(***********************************************************************************************************************************************
*********** OUTPUT FHPP DATA *******************************************************************************************************************
***********************************************************************************************************************************************)

pFHPP_DATA_OUT				:= ADR(FML_REF.FHPP.OUT);

IF FML_REF.Modbus THEN				// modbus word swapping
	//first 8 Byte
	FHPP_Target[0]			:= pFHPP_DATA_OUT^[1];
	FHPP_Target[1]			:= pFHPP_DATA_OUT^[0];
	FHPP_Target[2]			:= pFHPP_DATA_OUT^[3];
	FHPP_Target[3]			:= pFHPP_DATA_OUT^[2];
	IF FML_REF.HighByteFirst THEN	// high byte first (actual value2)
		FHPP_Target[4]		:= pFHPP_DATA_OUT^[6];
		FHPP_Target[5]		:= pFHPP_DATA_OUT^[7];
		FHPP_Target[6]		:= pFHPP_DATA_OUT^[4];
		FHPP_Target[7]		:= pFHPP_DATA_OUT^[5];
	ELSE							// low byte first (actual value2)
		FHPP_Target[4]		:= pFHPP_DATA_OUT^[5];
		FHPP_Target[5]		:= pFHPP_DATA_OUT^[4];
		FHPP_Target[6]		:= pFHPP_DATA_OUT^[7];
		FHPP_Target[7]		:= pFHPP_DATA_OUT^[6];
	END_IF	
	
	//second 8 Byte
	FHPP_Target[8]			:= pFHPP_DATA_OUT^[9];
	FHPP_Target[9]			:= pFHPP_DATA_OUT^[8];
	FHPP_Target[10]			:= pFHPP_DATA_OUT^[11];
	FHPP_Target[11]			:= pFHPP_DATA_OUT^[10];
	IF FML_REF.HighByteFirst THEN	// high byte first (actual value2)
		FHPP_Target[12]		:= pFHPP_DATA_OUT^[14];
		FHPP_Target[13]		:= pFHPP_DATA_OUT^[15];
		FHPP_Target[14]		:= pFHPP_DATA_OUT^[12];
		FHPP_Target[15]		:= pFHPP_DATA_OUT^[13];
	ELSE							// low byte first (actual value2)
		FHPP_Target[12]		:= pFHPP_DATA_OUT^[13];
		FHPP_Target[13]		:= pFHPP_DATA_OUT^[12];
		FHPP_Target[14]		:= pFHPP_DATA_OUT^[15];
		FHPP_Target[15]		:= pFHPP_DATA_OUT^[14];
	END_IF	
	
ELSE								//normal fieldbus: copy only
	// first 8 byte
	FHPP_Target[0]			:= pFHPP_DATA_OUT^[0];
	FHPP_Target[1]			:= pFHPP_DATA_OUT^[1];
	FHPP_Target[2]			:= pFHPP_DATA_OUT^[2];
	FHPP_Target[3]			:= pFHPP_DATA_OUT^[3];
	IF FML_REF.HighByteFirst THEN	// high byte first (actual value2)
		FHPP_Target[4]		:= pFHPP_DATA_OUT^[7];
		FHPP_Target[5]		:= pFHPP_DATA_OUT^[6];
		FHPP_Target[6]		:= pFHPP_DATA_OUT^[5];
		FHPP_Target[7]		:= pFHPP_DATA_OUT^[4];
	ELSE							// low byte first (actual value2)
		FHPP_Target[4]		:= pFHPP_DATA_OUT^[4];
		FHPP_Target[5]		:= pFHPP_DATA_OUT^[5];
		FHPP_Target[6]		:= pFHPP_DATA_OUT^[6];
		FHPP_Target[7]		:= pFHPP_DATA_OUT^[7];
	END_IF	
	
	// second 8 byte
	FHPP_Target[8]			:= pFHPP_DATA_OUT^[8];
	FHPP_Target[9]			:= pFHPP_DATA_OUT^[9];
	FHPP_Target[10]			:= pFHPP_DATA_OUT^[10];
	FHPP_Target[11]			:= pFHPP_DATA_OUT^[11];
	IF FML_REF.HighByteFirst THEN	// high byte first (actual value2)
		FHPP_Target[12]		:= pFHPP_DATA_OUT^[15];
		FHPP_Target[13]		:= pFHPP_DATA_OUT^[14];
		FHPP_Target[14]		:= pFHPP_DATA_OUT^[13];
		FHPP_Target[15]		:= pFHPP_DATA_OUT^[12];
	ELSE							// low byte first (actual value2)
		FHPP_Target[12]		:= pFHPP_DATA_OUT^[12];
		FHPP_Target[13]		:= pFHPP_DATA_OUT^[13];
		FHPP_Target[14]		:= pFHPP_DATA_OUT^[14];
		FHPP_Target[15]		:= pFHPP_DATA_OUT^[15];
	END_IF	
END_IF

(* ===== end of function block ============================= *)

END_FUNCTION_BLOCK

// Blocks/Parameterize/FPC_DATA_OBJECT
(* ============================================================================
   FESTO AG  Co., Esslingen - Copyright (c) 2015. All rights reserved.                       
 ------------------------------------------------------------------------------
 Functionblock:  FPC_DATA_OBJECT  
 Description:    function block to pass internal data objects to the controller
 Version:        V3.5.4.4        
 Composer:       bejk
 Last Update:    13.11.2017                                                                           
 ------------------------------------------------------------------------------ *)
{library private}
(* ----------------------------------------------------------------------------
Date        Name                Activity                                                                              
02.02.2010  Benjamin Kilgus     created
02.07.2013  Rudolf Schenke      Busy state and some other value clear
22.06.2015	Christian Hammer	adaptation to use this FB for all drives
04.09.2015  Christian Hammer	error handling (deleted RETVAL, created Status)
29.02.2016	Christian Hammer	set outputs to zero if not execute
13.11.2017	Christian Hammer	added blockade of FB for SFC-DC and MTR-DCI controller
=============================================================================== *)
{library public}

(* use this function block only with the function blocks FML_Read and FML_Write *)

FUNCTION_BLOCK FPC_DATA_OBJECT

VAR_IN_OUT
	FML_REF				: DT_FML_REF;		// structure of the parameter to control and parametrize the motorcontroller
END_VAR

VAR_INPUT
	Execute				: BOOL;  			// perfrom data exchange
	Write				: BOOL;  			// read or write the parameter (1=write / 0=read)
	Object				: INT; 				// number of internal data object
	Subindex			: INT; 				// subindex of the parameter to exchange
	Value				: DINT; 			// set value of internal data objects
END_VAR
VAR_OUTPUT
	Done				: BOOL; 			// transmission done
	Error				: BOOL; 			// transmission fault
	Status				: DT_FML_STATUS;	// structure with the status information of the function block and FPC
	ActObject			: INT;				// actual number of internal data objects
	ActSubindex			: DINT; 			// actual subindex of the parameter
	ActValue			: DINT; 			// actual value of internal data objects	
END_VAR

{library private}
VAR
	bInit           	: BOOL	:=FALSE;	// status of inizialisation of the FB
	lMemberID   		: INT;				// local member ID of the FB
	Step				: INT	:= 0;		// step number of the state machine

	TONInst				: TON;				// timer instance to monitor a timeout of the function block
	TimeStart			: BOOL;				// variable to start the timer instance
	TimeoutTime			: TIME := T#3S;		// timeout time 			
END_VAR
{library public}

(* ====== initial block routine ===================================== *)
(* ----- get MemberID for this function block ------------------------*)

IF NOT bInit THEN
	FML_REF.MemberIDmax		:= FML_REF.MemberIDmax +1;
	lMemberID				:= FML_REF.MemberIDmax;
	bInit					:= TRUE;
	Status.Err:=FALSE; Status.Cat:=FML_function_block; Status.ID:=FML_init_active;
END_IF

	
(* ====== supervision of timeout ==================================== *)
(* ----- timer to monitor a timeout of the function block ------------*)
TONInst(IN := TimeStart, PT := TimeoutTime);
IF TONInst.Q THEN
	Status.Err:=TRUE; Status.Cat:=FML_function_block; Status.ID:=FML_fb_timeout;
	Done					:= TRUE;
	Step					:= 100;
END_IF		

// this function block is not usable with SFC-DC and MTR-DCI
IF Execute 
	AND	((FML_REF.DeviceType = SFC_DC)
	OR (FML_REF.DeviceType = MTR_DCI)) THEN
		Done				:= TRUE;
		Status.Err:=TRUE; Status.Cat:=FML_function_block; Status.ID:=FML_wrong_device;
		Step				:= 100;
END_IF

(* ===== logic part ================================================= *)

IF NOT Execute AND (Step <> 0) THEN
 	FML_REF.MemberID		:= 0;
	FML_REF.ReqID			:= FML_FPC_REQ_none;
	FML_REF.FPCC_Modus		:= 0;
	FML_REF.PNU				:= 0;
	FML_REF.Subindex		:= 0;
	FML_REF.Value			:= 0;
	ActObject				:= 0;
	ActSubindex				:= 0;	
	ActValue				:= 0;
			
	Step					:= 0;
END_IF;

CASE Step OF
	0:(* *)
		Done				:= FALSE;
		TimeStart			:= FALSE;
		Status.Err:=FALSE; Status.Cat:=FML_no_category; Status.ID:=FML_no_error;

		IF (FML_REF.MemberID = 0) AND Execute THEN
    		FML_REF.MemberID		:= lMemberID;
			FML_REF.ReqID			:= FML_FPC_REQ_none;	
			FML_REF.PNU				:= 0;
			FML_REF.Subindex		:= 0;
			FML_REF.Value			:= 0;
			Status.Err:=FALSE; Status.Cat:=FML_function_block; Status.ID:=FML_fb_busy;
			
			IF (FML_REF.DeviceType = CMMP_AS) 
			OR (FML_REF.DeviceType = CMMS_AS) 
			OR (FML_REF.DeviceType = CMMS_ST)
			OR (FML_REF.DeviceType = CMMD_AS) THEN					(* CMMP-AS or CMMS_AS or CMMS_ST or CMMD_AS *)
				FML_REF.FPCC_Modus	:= FML_FPC_MODUS_PNU_11BIT;		// FPC standard
				Step				:= 10;				
			ELSE 													(* CMMO-ST AND EMCA-EC *)
				FML_REF.FPCC_Modus	:= FML_FPC_MODUS_DATA_OBJECT;	// EPC access for internal data objects
				Step				:= 20;
			END_IF
			
		ELSIF (FML_REF.MemberID <> lMemberId) AND Execute THEN
			Status.Err:=FALSE; Status.Cat:=FML_function_block; Status.ID:=FML_other_fb_active;
		END_IF

(* CMMP-AS or CMMS_AS or CMMS_ST or CMMD_AS or SFC_DC or MTR_DCI *)		
	10:(* open tunnel access *)
		FML_REF.ReqID				:= FML_FPC_REQ_write_array_dword; 
		FML_REF.PNU					:= 80;
		FML_REF.Subindex			:= 1;
		FML_REF.Value				:= Object;
		TimeStart					:= TRUE;
		
		IF FML_REF.Done AND NOT FML_REF.Err THEN
			TimeStart				:= FALSE;
      		FML_REF.ReqID         	:= FML_FPC_REQ_none;  
      		Step                  	:= 11;
  		(* error occured *)
  		ELSIF FML_REF.Done AND FML_REF.Err THEN
			TimeStart				:= FALSE;      		
      		Step                 	:= 30;
 		END_IF


	11:(* access granted *)
		TimeStart					:= TRUE;
	
		IF NOT FML_REF.Done THEN
			TimeStart				:= FALSE;
			(* write internal data objects *)
			IF Write THEN
				FML_REF.ReqID			:= FML_FPC_REQ_write_array_dword; 
				FML_REF.PNU				:= 82;
				FML_REF.Subindex		:= 1;
				FML_REF.Value			:= Value;
				Step					:= 30;
    		(* read internal data objects *)
			ELSE
				FML_REF.ReqID			:= FML_FPC_REQ_read_array;	  
				FML_REF.PNU				:= 81;
				FML_REF.Subindex		:= 1;
				FML_REF.Value			:= 0;
				Step					:= 30;
			END_IF
		END_IF
		
(* CMMO-ST AND EMCA-EC *)
	20:		
		IF Write THEN
			FML_REF.ReqID			:= FML_FPC_REQ_write_array_dword; 
		ELSE
			FML_REF.ReqID			:= FML_FPC_REQ_read_array;
		END_IF	
			
		FML_REF.PNU					:= Object;
		FML_REF.Subindex			:= Subindex;
		FML_REF.Value				:= Value;
		Step						:= 30;

	30:(* set output variables *)
		TimeStart					:= TRUE;
		
		IF FML_REF.Done THEN
			FML_REF.ReqID			:= FML_FPC_REQ_none;
			TimeStart				:= FALSE;
			Done					:= TRUE;
			Step					:= 100;
			
			IF FML_REF.Err THEN
				Status.Err:=TRUE; Status.Cat:=FML_parameter_transfer; Status.ID:=FML_REF.ActValue;
				ActValue			:= 0;
				ActSubindex			:= 0;
				ActObject			:= 0;   
			ELSE
				Status.Err:=FALSE; Status.Cat:=FML_no_category; Status.ID:=FML_no_error;
				
				IF (FML_REF.DeviceType = CMMP_AS) 
				OR (FML_REF.DeviceType = CMMS_AS) 
				OR (FML_REF.DeviceType = CMMS_ST)
				OR (FML_REF.DeviceType = CMMD_AS) 
				OR (FML_REF.DeviceType = SFC_DC) 
				OR (FML_REF.DeviceType = MTR_DCI) THEN					(* CMMP-AS or CMMS_AS or CMMS_ST or CMMD_AS or SFC_DC or MTR_DCI *)
					ActObject			:= Object;
					ActSubindex			:= Subindex;
					ActValue			:= FML_REF.ActValue;			
				ELSE 												(* CMMO-ST AND EMCA-EC *)
					ActObject			:= FML_REF.ActPNU;
					ActSubindex			:= FML_REF.ActSubindex;
					ActValue			:= FML_REF.ActValue;
				END_IF
			END_IF
  		END_IF
	
	100: (* done - do nothing *)
		;
		
END_CASE

Status.Msg					:= GetStatusMessage(Status);
Error						:= Status.Err;

(* ===== end of function block ============================= *)

END_FUNCTION_BLOCK

// Blocks/Parameterize/FPC_DIAG
(* ============================================================================
   FESTO AG & Co. KG, Esslingen - Copyright (c) 2015. All rights reserved.                       

 Functionblock:  FPC_DIAG
 Description:    function block to read the most actual error
 Version:        V3.5.7.21         
 Composer:       bejk
 Date:           13.11.2017                                                                           
------------------------------------------------------------------------------- *)
{library private}
(* ----------------------------------------------------------------------------
Date        Name             	Activity                                                                              
01.04.2014  Benjamin Kilgus  	V3.1  created out of CMMS_AS_PRM_SINGLE
09.02.2015  Rudolf Schenke   	Implement 16-bit mode with hide preset
22.06.2015	Christian Hammer	adaptation to use this FB for all drives
04.09.2015  Christian Hammer	error handling (deleted RETVAL, created Status)
13.11.2017	Christian Hammer	added blockade of FB for SFC-DC and MTR-DCI controller
=============================================================================== *)
{library public}

(* use this function block only with the function blocks FML_Read and FML_Write *)

FUNCTION_BLOCK FPC_DIAG

VAR_IN_OUT
	FML_REF        		: DT_FML_REF;		// structure of the parameter to control and parametrize the motorcontroller
END_VAR

VAR_INPUT															
	Execute         	: BOOL;  			// perfrom data exchange
END_VAR

VAR_OUTPUT
	Done            	: BOOL;  			// execution done
	Error				: BOOL; 			// transmission fault
	Status				: DT_FML_STATUS;	// structure with the status information of the function block and FPC	
	MessageNumber   	: INT;  			// fault occured
	MessageDescription  : STRING;			// discription of the error
END_VAR

{library private}
VAR
	bInit           	: BOOL	:=FALSE;	// status of inizialisation of the FB
	lMemberID   		: INT;				// local member ID of the FB	
	
	TONInst				: TON;				// timer instance to monitor a timeout of the function block
	TimeStart			: BOOL;				// variable to start the timer instance
	TimeoutTime			: TIME := T#3S;		// timeout time 
END_VAR
{library public}

(* ====== initial block routine ===================================== *)
(* ----- get MemberID for this function block ------------------------*)
IF NOT bInit THEN
	FML_REF.MemberIDmax		:= FML_REF.MemberIDmax +1;
	lMemberID            	:= FML_REF.MemberIDmax;
	bInit              		:= TRUE;
	Status.Err:=FALSE; Status.Cat:=FML_function_block; Status.ID:=FML_init_active;
END_IF


(* ====== supervision of timeout ==================================== *)
(* ----- timer to monitor a timeout of the function block ------------*)
TONInst(IN := TimeStart, PT := TimeoutTime);
IF TONInst.Q THEN
	Done					:= TRUE;
	Status.Err:=TRUE; Status.Cat:=FML_function_block; Status.ID:=FML_fb_timeout;
END_IF					

	
(* ===== logic part ================================================= *)
(* ----- ASSIGNMENT OF STATUS --------------------------------------- *)
// this function block is not usable with SFC-DC and MTR-DCI
IF ((FML_REF.DeviceType = SFC_DC)
OR (FML_REF.DeviceType = MTR_DCI)) THEN
	IF Execute THEN
		Done					:= TRUE;
		Status.Err:=TRUE; Status.Cat:=FML_function_block; Status.ID:=FML_wrong_device;
	ELSE
		Done					:= FALSE;
		Status.Err:=FALSE; Status.Cat:=FML_no_category; Status.ID:=FML_no_error;
	END_IF
	
ELSE
	IF FML_REF.MemberID = lMemberId THEN
		IF FML_REF.Done AND NOT FML_REF.Err AND NOT Status.Err THEN
			Done              	:= TRUE;
			TimeStart			:= FALSE;
			
			IF FML_REF.ActValue = 65535 THEN 			// special: -1 to 0
				MessageNumber 	:= 0; 
			ELSE
				MessageNumber	:= DINT_TO_INT(FML_REF.ActValue);	
			END_IF  
			
			MessageDescription	:= FaultString(MessageNumber, FML_REF.DeviceType);
			Status.Err:=FALSE; Status.Cat:=FML_no_category; Status.ID:=FML_no_error;
			
		ELSIF FML_REF.Err THEN
			Status.Err:=TRUE; Status.Cat:=FML_parameter_transfer; Status.ID:=FML_REF.ActValue;
		END_IF
	END_IF
	
	(* ----- ASSIGNMENT OF CONTROL at rising edge of Execute ------------ *)
	IF (FML_REF.MemberID = 0) AND Execute THEN
		TimeStart				:= TRUE;
		Status.Err:=FALSE; Status.Cat:=FML_function_block; Status.ID:=FML_fb_busy;
		FML_REF.MemberID    	:= lMemberID;
		FML_REF.ReqID			:= FML_FPC_REQ_read_array;
	 
		IF (FML_REF.DeviceType = CMMP_AS) 
		OR (FML_REF.DeviceType = CMMS_AS) 
		OR (FML_REF.DeviceType = CMMS_ST)
		OR (FML_REF.DeviceType = CMMD_AS) THEN					(* CMMP-AS or CMMS_AS or CMMS_ST or CMMD_AS *)
			FML_REF.FPCC_Modus 	:= E_FML_FPC_MODUS.FML_FPC_MODUS_PNU_11BIT;
			FML_REF.PNU			:= 201;
			FML_REF.Subindex	:= 1;
	
		ELSE 													(*******EMCA-EC or CMMO-ST*******)	
			FML_REF.FPCC_Modus 	:= E_FML_FPC_MODUS.FML_FPC_MODUS_PNU_16BIT;
			FML_REF.PNU			:= 205;
			FML_REF.Subindex	:= 1;
		END_IF
		FML_REF.Value			:= 0;
	
	ELSIF (FML_REF.MemberID = lMemberId) AND NOT Execute THEN
		FML_REF.ReqID			:= FML_FPC_REQ_none;
		FML_REF.PNU				:= 0;
		FML_REF.Subindex		:= 0;
		FML_REF.Value			:= 0;
		MessageNumber			:= 0;
		MessageDescription		:= '';
		TimeStart				:= TRUE;
		IF NOT FML_REF.Done THEN
			FML_REF.MemberID	:= 0;     				// free the modul after all transmission
			TimeStart			:= FALSE;
			Done				:= FALSE;
			Status.Err:=FALSE; Status.Cat:=FML_no_category; Status.ID:=FML_no_error;
		END_IF;
		
	ELSIF (FML_REF.MemberID <> lMemberId) THEN
		IF Execute THEN
			Status.Err:=FALSE; Status.Cat:=FML_function_block; Status.ID:=FML_other_fb_active;
		ELSE
			Status.Err:=FALSE; Status.Cat:=FML_no_category; Status.ID:=FML_no_error;
		END_IF 
	END_IF
END_IF

Status.Msg						:= GetStatusMessage(Status);
Error							:= Status.Err;

(* ===== end of function block ============================= *)

END_FUNCTION_BLOCK

// Blocks/Parameterize/FPC_FILE_ARRAY
(* ============================================================================
   FESTO AG & Co. KG, Esslingen - Copyright 2015. All rights reserved.                       
 ------------------------------------------------------------------------------
 Functionblock: PRM_FILE_ARRAY
 Description:   function block to save and restore parameter file in a array
                  - Upload: from controller to PLC (array)
                  - Download: from PLC (array) to controller 
 ------------------------------------------------------------------------------
 Version:        V3.5.7.22         
 Composer:       bejk 
 Last Update:    25.04.2018                                                                              
 ------------------------------------------------------------------------------ *)
{library private}
(* ----------------------------------------------------------------------------
 Date       Name             	Activity                                                                              
 01.04.2014 Benjamin Kilgus  	created
 07.09.2014 Rudolf Schenke   	NextSequence() for Sequence++ created
                             	Correct all compiler warning causes 
                             	Set the fix directory name to 'CMMOparameter'
                             	Download: More direct buffer management
 14.09.2014 Rudolf Schenke   	VIS_CMMO_PRM_FILE prepared and adapted
 29.09.2014 Rudolf Schenke   	Redesign from file functions to file FBs
 10.12.2014 Rudolf Schenke   	Redesign der Schnittstelle zum file FB 
 14.01.2015 Rudolf Schenke   	Fehler bei Create Directory korrigiert (173989)
 09.03.2015 Rudolf Schenke   	CMMO_PRM_FILE: Umstellung auf neue IODD für IO-Link                              
 22.06.2015	Christian Hammer	adaptation to use this FB for all drives	
 29.02.2016	Christian Hammer	changed Line 265 (IF Status.ID==FML_par_file_err)
 20.10.2017 Christian Hammer	device type "CMMP_AS" added (deleted in line 12)
 13.11.2017	Christian Hammer	added blockade of FB for SFC-DC and MTR-DCI controller
 25.04.2018 Benjamin Klein		added blockade of FB for CMXH-ST controller
=============================================================================== *)
{library public}

(* use this function block only with the function blocks FML_Read and FML_Write *)

FUNCTION_BLOCK FPC_FILE_ARRAY

VAR_IN_OUT
	FML_REF    		: DT_FML_REF;			// structure of the parameter to control and parametrize the motorcontroller
END_VAR

VAR_INPUT
	Execute     	: BOOL;     			// perform data exchange	
	Upload 			: BOOL;	    			// upload operation
	Download    	: BOOL;     			// download operation
	SizeOfFileArray : UINT;           		// size of the file array
	AdrOfFileArray  : POINTER TO BYTE; 		// 1. element of file array
END_VAR

VAR_OUTPUT
	Done        	: BOOL;  				// transmission done 
	Error			: BOOL; 				// error during execution	
	Status			: DT_FML_STATUS;		// structure with the status information of the function block	
	CountByte		: DINT;        			// dynamic byte counter
	FileSize		: DINT;	        		// resulting file size
END_VAR		

{library private}

VAR CONSTANT
 	udLength			: INT := 6;			// length of a file token
	ArrayWithZeros		: ARRAY[0..5] OF BYTE := [udLength(0)]; 			//[0,0,0,0,0,0]
END_VAR

VAR
	//general variables
	bInit      			: BOOL := FALSE;	// init flag
	lMemberID     		: INT;
	SendRepeat			: INT;
	Sequence			: INT;   			// sequence counter (incremented after each transfer)
	Step				: INT;      		// state machine

	//buffer
	pbyBuffer			: POINTER TO ARRAY [1..udLength] OF BYTE;
	Buffer				: ARRAY [1..udLength] OF BYTE := [udLength(0)]; 	//[0,0,0,0,0,0]
	PtrToDataFileArray  : POINTER TO BYTE;
	i					: INT;
		
	// visu
	vis_upload			: BOOL;   			// upload active for visu
	vis_download		: BOOL;  			// download active for visu

	//timout
	TimeStart			: BOOL;
	TimeStop			: BOOL;
 	TONInst				: TON;
END_VAR
{library public}

(* ====== initial block routine ===================================== *)
(* ----- get MemberID for this function block ------------------------*)
IF NOT bInit THEN
	FML_REF.MemberIDmax		:= FML_REF.MemberIDmax +1;
	lMemberID            	:= FML_REF.MemberIDmax;
	bInit              		:= TRUE;
	Status.Err:=FALSE; Status.Cat:=FML_function_block; Status.ID:=FML_init_active;
END_IF

//no file transfer in CMMS_AS or CMMS_ST or CMMD_AS
IF Execute 
	AND ((FML_REF.DeviceType = CMMS_AS) 
		OR (FML_REF.DeviceType = CMMS_ST)
		OR (FML_REF.DeviceType = CMMD_AS)
		OR (FML_REF.DeviceType = SFC_DC)
		OR (FML_REF.DeviceType = MTR_DCI)
		OR (FML_REF.DeviceType = CMXH_ST)) THEN
			Done				:= TRUE;
			Status.Err:=TRUE; Status.Cat:=FML_function_block; Status.ID:=FML_wrong_device;
			Step				:= 27;
END_IF


(* ===== logic part ================================================= *)
IF NOT Execute AND (Step <> 0) THEN 										// reset all parameter (also bus data)
	FML_REF.MemberID     				:= 0;
	FML_REF.ReqID      	    			:= FML_FPC_REQ_none;
	FML_REF.FPCC_Modus					:= 0;
	FML_REF.FPCC_Packet.Control			:= 0;
	FML_REF.FPCC_Packet.BitSequenceNr	:= 0;
	FML_REF.FPCC_Packet.Data			:= ArrayWithZeros;
			
	Step 								:= 0;
END_IF

TONInst(IN := TimeStart, PT := T#3S, Q => TimeStop);						//timer for timeout


CASE Step OF 
	0:(* initial prepare*)
		Done			:= FALSE;
		Sequence		:= 0;
		CountByte 		:= 0;
		FileSize		:= 0;
		vis_download	:= FALSE;
		vis_upload		:= FALSE;
		SendRepeat		:= 0;
		Status.Err:=FALSE; Status.Cat:=FML_no_category; Status.ID:=FML_no_error;
    
		IF Execute AND FML_REF.MemberID = 0 THEN							// parameterchannel is free
			FML_REF.MemberID   		:= lMemberID;
			FML_REF.ReqID			:= FML_FPC_REQ_none;
					  
    		// check for double mode selection by visu
			IF NOT (Upload XOR Download) THEN  								// both or none are selected -> error
 				Status.Err:=TRUE; Status.Cat:=FML_parameter_transfer; Status.ID:=FML_direction_err;
				Step				:= 27;
       			RETURN;
			
			ELSIF Upload AND NOT Download THEN
				pbyBuffer			:= ADR(FML_REF.FPCS_Packet.Data);
				PtrToDataFileArray	:= AdrOfFileArray;
				vis_upload 			:= TRUE;
				Status.Err:=FALSE; Status.Cat:=FML_function_block; Status.ID:=FML_fb_busy;  	// execute starts here				
				Step 				:= 1;														// step 1 = starts upload
			
			ELSIF Download AND NOT Upload THEN
				pbyBuffer 	  		:= ADR(Buffer);
				PtrToDataFileArray	:= AdrOfFileArray;
				vis_download		:= TRUE;
				Status.Err:=FALSE; Status.Cat:=FML_function_block; Status.ID:=FML_fb_busy; 		// execute starts here
				Step 				:= 6;														// step 6 = starts download
			END_IF

	  	  // other FB active 
		ELSIF Execute AND FML_REF.MemberID <> lMemberId THEN
			Status.Err:=FALSE; Status.Cat:=FML_function_block; Status.ID:=FML_other_fb_active; 		
		END_IF
		
		
    //===== upload handling ===============
	1: (*start requirement - upload*)
		FML_REF.FPCC_Modus 			    	:= 4;							// choose mode
		FML_REF.ReqID 						:= FML_FPC_REQ_read_file; 		// upload
		FML_REF.FPCC_Packet.Control			:= FML_FPC_FILE_TRANSFER_start; // start transmission
		FML_REF.FPCC_Packet.BitSequenceNr	:= Sequence;
		FML_REF.FPCC_Packet.Data			:= Buffer; 						// user data are zero
		TimeStart 							:= TRUE; 						// start timer for timeout
		Step 								:= 2;
		
	2: (*wait for response from controller - upload*)
		// controller also sends upload data with the size of the parameter file
		IF FML_REF.RespID = FML_FPC_RESP_file_done AND FML_REF.FPCS_Packet.Control = FML_REF.FPCC_Packet.Control AND FML_REF.FPCS_Packet.BitSequenceNr = Sequence THEN
			Buffer							:= FML_REF.FPCS_Packet.Data;	// write incoming data from controller into buffer (6 Byte)
			FOR i := 0 TO 5 DO
				PtrToDataFileArray^			:= Buffer[i+1];					// write data from buffer to output (each byte separately)
				PtrToDataFileArray			:= PtrToDataFileArray + 1;
			END_FOR
			
			IF Sequence = 0 THEN 											// save size of parameterfile
				CalculateFilesize();  										// calculate size of file as a multiple of udLength	
				
				IF FileSize > SizeOfFileArray THEN							// check if the array is big enough
					Step 			    	:= 27; 							// array is to small --> error state
					Status.Err:=TRUE; Status.Cat:=FML_parameter_transfer; Status.ID:=FML_volume_err;
					RETURN;
				END_IF
			END_IF
		 	
			CountByte 						:= CountByte + udLength;		// count up the bytes
			NextSequence();													// count up the sequence
			TimeStart 						:= FALSE; 						// reset timer
			Step 							:= 3;
			
		ELSE //---- timeout ----
			IF TimeStop THEN
				TimeStart 					:= FALSE; 						// reset timer
				Step 						:= 4; 							// start acknowledgment is missing -->  check Step 4 on error
			END_IF
		END_IF

	3: (*request package - upload*)
		FML_REF.FPCC_Packet.Control 		:= FML_FPC_FILE_TRANSFER_active;
		FML_REF.FPCC_Packet.BitSequenceNr 	:= Sequence;
		FML_REF.FPCC_Packet.Data 			:= Buffer;		
		Step 								:= 4;

	4: (*wait for answer - upload*)
		TimeStart 							:= TRUE; 						// restart timer fot timeout (for each packet)
		// expect and save packet
		IF FML_REF.RespID = FML_FPC_RESP_file_done AND FML_REF.FPCS_Packet.Control = FML_REF.FPCC_Packet.Control AND FML_REF.FPCS_Packet.BitSequenceNr = Sequence THEN
			Buffer							:= FML_REF.FPCS_Packet.Data;	// write incoming data from controller into buffer (6 Byte)
			FOR i := 0 TO 5 DO
				PtrToDataFileArray^			:= Buffer[i+1];					// write data from buffer to output (each byte separately)
				PtrToDataFileArray			:= PtrToDataFileArray + 1;
			END_FOR
			
			CountByte 						:= CountByte + udLength;		// count up the bytes
			NextSequence();       											// count sequence
			TimeStart						:= FALSE;
			Step							:= 3; 
		
		// finish upload, controller sends stopp
		ELSIF FML_REF.RespID = FML_FPC_RESP_file_done AND FML_REF.FPCS_Packet.Control = FML_FPC_FILE_TRANSFER_stop AND FML_REF.FPCS_Packet.BitSequenceNr = Sequence THEN
			TimeStart 						:= FALSE;
			IF CountByte <> Filesize OR CountByte < 100 THEN 				// check if all bytes are uploaded
				Step 			    		:= 21; 							// wrong size --> error state
				Status.Err:=TRUE; Status.Cat:=FML_parameter_transfer; Status.ID:=FML_incomplete; 
			ELSE
				Step 			    		:= 20;							// size is right, upload successful, end state		
			END_IF
						
		// error from controller, general EFPC error
		ELSIF FML_REF.RespID = FML_FPC_RESP_error THEN
			Status.Err:=TRUE; Status.Cat:=FML_parameter_transfer; Status.ID:=FML_REF.FPCS_Packet.Data[1]+1000; 
			TimeStart 						:= FALSE;
			NextSequence();     											// count sequence modul
			Step 			  				:= 23;  						// send stopp after error
			
		// error from controller - upload
		ELSIF FML_REF.FPCS_Packet.Control = FML_FPC_FILE_TRANSFER_error THEN
			Status.Err:=TRUE; Status.Cat:=FML_parameter_transfer; Status.ID:=FML_REF.FPCS_Packet.Data[1]+1000; 	// get error code from data at byte 1
			TimeStart						:= FALSE;
			NextSequence();     											// count sequence modulo
			Step							:= 23;  						// send stopp after error	
		
		ELSE 
			//timeout
			IF TimeStop THEN
				Status.Err:=TRUE; Status.Cat:=FML_parameter_transfer; Status.ID:=FML_time_out; 
				Step						:= 21;  						// send error message to controller
				TimeStart					:= FALSE;
			END_IF	
		END_IF
	
	6: (*start requirement - download*)
		FOR i := 0 TO 5 DO
			Buffer[i+1]						:= PtrToDataFileArray^;			// write data from data array (input) into buffer (each byte separately)
			PtrToDataFileArray				:= PtrToDataFileArray + 1;
		END_FOR

		IF Sequence = 0 THEN    											
			CalculateFilesize(); 											// calculate size of file as a multiple of udLength
			
			IF FileSize < 262 THEN  										// file larger than header --> error
				Step 						:= 27;
				Status.Err:=TRUE; Status.Cat:=FML_parameter_transfer; Status.ID:=FML_size_err; 
				RETURN;
			ELSIF FileSize > SizeOfFileArray THEN							// check if the array is big enough
				Step 			    		:= 27; 							// array is to small --> error state
				Status.Err:=TRUE; Status.Cat:=FML_parameter_transfer; Status.ID:=FML_volume_err;
				RETURN;
			END_IF
		END_IF	
				
		FML_REF.FPCC_Packet.Data 			:= Buffer;						// write data from buffer to controller (6 byte)	
		CountByte 							:= CountByte + udLength;
		FML_REF.FPCC_Modus					:= 4;							// modus parameter file 
		FML_REF.ReqID						:= FML_FPC_REQ_write_file; 		// download
		FML_REF.FPCC_Packet.Control			:= FML_FPC_FILE_TRANSFER_start; // start transfer
		FML_REF.FPCC_Packet.BitSequenceNr	:= Sequence;
		TimeStart 							:= TRUE;
		Step 								:= 7;

			
	7: (*wait for response from controller - download*)
		IF FML_REF.RespID = FML_FPC_RESP_file_done AND FML_REF.FPCS_Packet.Control = FML_REF.FPCC_Packet.Control AND FML_REF.FPCS_Packet.BitSequenceNr = Sequence THEN
			Sequence 						:= 1;
			Step 							:= 8;
		ELSE
			//timeout
			IF TimeStop THEN
				TimeStart 					:= FALSE;
				Step 						:= 9;
			END_IF
		END_IF

	8: (*send packet - download*)
		IF CountByte < FileSize THEN
			FOR i := 0 TO 5 DO
				Buffer[i+1]					:= PtrToDataFileArray^;			// write data from data array (input) into buffer (each byte separately)
			PtrToDataFileArray				:= PtrToDataFileArray + 1;
		END_FOR
		
		FML_REF.FPCC_Packet.Data 				:= Buffer;					// write data from buffer to controller (6 byte)
			CountByte							:= CountByte + udLength;
			FML_REF.FPCC_Packet.Control			:= FML_FPC_FILE_TRANSFER_active;
			FML_REF.FPCC_Packet.BitSequenceNr	:= Sequence;
			Step								:= 9;
				
		ELSE          //---- end of file detected -ä stop to device
			FML_REF.FPCC_Packet.Control 		:= FML_FPC_FILE_TRANSFER_stop;
			FML_REF.FPCC_Packet.BitSequenceNr	:= Sequence;
			FML_REF.FPCC_Packet.Data 			:= Buffer;
			Step								:= 9;
		END_IF
	
	9: (*wait for confirmation of receipt of controller - download*)
		// receive and process message 
		TimeStart								:= TRUE;
		IF FML_REF.RespID = FML_FPC_RESP_file_done AND FML_REF.FPCS_Packet.Control = FML_FPC_FILE_TRANSFER_active AND FML_REF.FPCS_Packet.BitSequenceNr = Sequence THEN
			NextSequence();														// count sequence modulo
			TimeStart							:= FALSE;       												
			Step								:= 8;
			
		// if stop has been sent to the controller
		ELSIF FML_REF.RespID = FML_FPC_RESP_file_done AND FML_REF.FPCS_Packet.Control = FML_FPC_FILE_TRANSFER_stop AND FML_REF.FPCS_Packet.BitSequenceNr = Sequence THEN
			IF CountByte <> Filesize OR CountByte < 100 THEN 					// check if parameterfile has been loaded
				Step 			:= 21; 											// wrong size, error step
				Status.Err:=TRUE; Status.Cat:=FML_parameter_transfer; Status.ID:=FML_incomplete;
			ELSE
				Step 			:= 20;											// right size, download successful, end state    // check if all bytes are uploaded
			END_IF
			TimeStart 			:= FALSE;
			
		// error from controller, general EFPC error
		ELSIF FML_REF.RespID = FML_FPC_RESP_error THEN
			Status.Err:=TRUE; Status.Cat:=FML_parameter_transfer; Status.ID:=FML_REF.FPCS_Packet.Data[1]+1000;	// get error code from data at byte 1
			NextSequence();       												// count sequence modulo
			Step				:= 23;
			TimeStart 			:= FALSE;
			
		// error form controller - Download
		ELSIF FML_REF.FPCS_Packet.Control = FML_FPC_FILE_TRANSFER_error THEN
			Status.Err:=TRUE; Status.Cat:=FML_parameter_transfer; Status.ID:=FML_REF.FPCS_Packet.Data[1]+1000;	// get error code from data at byte 1
      		NextSequence();       												// count sequence modulo
			IF Status.ID = FML_par_file_err THEN								// If Status.ID == 1008
				Step 			:= 27;
			ELSE
				Step 			:= 23;
			END_IF
			TimeStart 			:= FALSE;
		
		ELSE
			// timeout
			IF TimeStop THEN
				Status.Err:=TRUE; Status.Cat:=FML_parameter_transfer; Status.ID:=FML_time_out; 
				Step 			:= 21;
				TimeStart		:= FALSE;
			END_IF
		END_IF
	
	20:	(*  ==== done with no error ==== *)
		Status.Err:=FALSE; Status.Cat:=FML_no_category; Status.ID:=FML_no_error;
		Step					:= 27;      						// wait for NOT execute
	
		
	21: (*send error message to Controller*)
		NextSequence();      				 						// count sequence modulo
		FML_REF.FPCC_Modus 					:= 4;
		FML_REF.FPCC_Packet.Control 		:= 3;
		FML_REF.FPCC_Packet.BitSequenceNr  	:= Sequence;
		FML_REF.FPCC_Packet.Data 			:= Buffer;
		TimeStart							:= TRUE;
		Step 								:= 22;
			
	22: (*wait for error message from controller*)
		IF FML_REF.RespID = FML_FPC_RESP_file_done AND FML_REF.FPCS_Packet.Control = FML_FPC_FILE_TRANSFER_error THEN
			NextSequence();       									// count sequence modulo
			TimeStart						:= FALSE;
			Step 							:= 23;
		ELSE
			IF TimeStop THEN
				Status.Err:=TRUE; Status.Cat:=FML_parameter_transfer; Status.ID:=FML_time_out;
				TimeStart 					:= FALSE;
				Step 						:= 23;
			END_IF
		END_IF
		
	23: (*send STOPP after error*)	
		FML_REF.FPCC_Packet.Control 		:= 2; 					// after error STOPP is sending to Controller
		FML_REF.FPCC_Packet.BitSequenceNr 	:= Sequence;
		FML_REF.FPCC_Packet.Data 			:= Buffer;
		TimeStart 							:= TRUE;
		Step 								:= 24;		
		
	24: (*query wheater stop was confirmed by controller*)
		IF (FML_REF.RespID = FML_FPC_RESP_file_done AND FML_REF.FPCS_Packet.Control = 2) OR  FML_REF.RespID = 7 THEN
			Step 							:= 27;
			TimeStart 						:= FALSE;
		ELSIF FML_REF.RespID = FML_FPC_RESP_file_done AND FML_REF.FPCS_Packet.Control = 3 AND SendRepeat < 4 THEN
			Status.ID						:= FML_REF.FPCS_Packet.Data[1]+1000;			// get error code from data at byte 1
			IF Status.ID <> 1000 THEN
				Status.Err					:= TRUE;
				Status.Cat					:= FML_parameter_transfer;
			END_IF
			
			Sequence 						:= Sequence + 1;
			SendRepeat 						:= SendRepeat + 1;
			TimeStart 						:= FALSE;
			Step 							:= 23;
		ELSE
			// timeout
			IF TimeStop THEN
				Status.Err:=TRUE; Status.Cat:=FML_parameter_transfer; Status.ID:=FML_time_out;
				TimeStart 					:= FALSE;
				Step 						:= 27;
			END_IF
		END_IF
		
  
  27: (*idle - wait for execute = false*)
		vis_upload 							:= FALSE;
		vis_download 						:= FALSE;
		Done								:= TRUE;
		Step								:= 30;
    		
  30: (*do nothing - wait for NOT execute*)
    	;
  
END_CASE

Status.Msg				:= GetStatusMessage(Status);
Error					:= Status.Err;

(* ===== end of function block ============================= *)

ACTION CalculateFilesize:
(* -----------------------------------------------------
   This action calculates the file size as a couple of 6 
   from the first 2 bytes of the buffer
   ----------------------------------------------------- *)

 	FileSize	:= DWORD_TO_DINT( SHL(BYTE_TO_DWORD(pbyBuffer^[2]),8) OR pbyBuffer^[1]); 	// length of data field
	FileSize	:= (Filesize + 2 * udLength -1) / udLength ; 								// +6: size of parameter file at first position, +5 und /6 for rounding up 
	FileSize	:= FileSize * udLength; 													// bytesize is being computed out of number of packages
END_ACTION

ACTION NextSequence:
(* -----------------------------------------------------
   This action increments the Sequence counter modulo 32. 
   It is used at 8 points in CMMO_ST_PRM_FILE
   ----------------------------------------------------- *)
	IF Sequence = 31 THEN
		Sequence 	:= 0;
	ELSE
		Sequence 	:= Sequence + 1;
	END_IF
END_ACTION

END_FUNCTION_BLOCK

// Blocks/Parameterize/FPC_DIRMP
(* ============================================================================
   FESTO AG & Co. KG, Esslingen - Copyright 2015. All rights reserved.                       
 ------------------------------------------------------------------------------
 Functionblock:  PRM_DIRMP  
 Description:    function block to pass dynamic parameter values for direct-mode-positioncontrol
 Version:        V3.5.7.21        
 Composer:       bejk
 Last update:    13.11.2017                                                                           
------------------------------------------------------------------------------- *)
{library private}
(* -----------------------------------------------------------------------------
Date        Name            	Activity                                                                              
11.03.2009  Benjamin Kilgus 	created
            Rudolf Schenke  	PNU array created 
09.02.2015  Rudolf Schenke  	Implement 16-bit mode with hide preset 
22.06.2015	Christian Hammer	adaptation to use this FB for all drives
04.09.2015  Christian Hammer	error handling (deleted RETVAL, created Status)
13.11.2017	Christian Hammer	added blockade of FB for SFC-DC and MTR-DCI controller
=============================================================================== *)
{library public}

(* use this function block only with the function blocks FML_Read and FML_Write *)

FUNCTION_BLOCK FPC_DIRMP

VAR_IN_OUT
	FML_REF					: DT_FML_REF;		// structure of the parameter to control and parametrize the motorcontroller
END_VAR

VAR_INPUT
	Execute             	: BOOL;				// perfrom data exchange
	Write               	: BOOL;				// read or write the parameter	(1=write/0=read)
	Velocity            	: DINT;				// base velocity directmode positioning
	Acceleration			: DINT; 			// acceleration directmode positioning
 	Deceleration        	: DINT; 			// deceleration directmode positioning
END_VAR

VAR_OUTPUT	
	Done                	: BOOL;				// transmission done
	Error					: BOOL; 			// transmission fault
	Status					: DT_FML_STATUS;	// structure with the status information of the function block and FPC
	ActVelocity         	: DINT;  			// base velocity directmode positioning
	ActAcceleration     	: DINT;  			// acceleration directmode positioning
	ActDeceleration     	: DINT;  			// deceleration directmode positioning
END_VAR

{library private}
VAR
	bInit           		: BOOL	:=FALSE;										// status of inizialisation of the FB
	lMemberID   			: INT;													// local member ID of the FB													
	Param       			: ARRAY [1..maxParamCount] OF DT_FML_PRM_DESCRIPTION;	// parameter to write in motorcontroller
	listPNU    				: ARRAY [1..maxParamCount] OF INT := [540,541,542];		// PNUs for the parameter 
	Step        			: INT:= 0; 												// actual step number 
	ixPar       			: INT:= 1;  											// index for the array

	TONInst					: TON;													// timer instance to monitor a timeout of the function block
	TimeStart				: BOOL;													// variable to start the timer instance
	TimeoutTime				: TIME := T#3S;											// timeout time 	
END_VAR

VAR CONSTANT
	maxParamCount			: INT := 3;												// max number of the parameter 
END_VAR

{library public}

(* ====== initial block routine ===================================== *)
(* ----- get MemberID for this function block ------------------------*)
IF NOT bInit THEN
	FML_REF.MemberIDmax		:= FML_REF.MemberIDmax +1;
	lMemberID				:= FML_REF.MemberIDmax;
	bInit					:= TRUE;
	Status.Err:=FALSE; Status.Cat:=FML_function_block; Status.ID:=FML_init_active;
END_IF


(* ====== supervision of timeout ==================================== *)
(* ----- timer to monitor a timeout of the function block ------------*)
TONInst(IN := TimeStart, PT := TimeoutTime);
IF TONInst.Q THEN
	Status.Err:=TRUE; Status.Cat:=FML_function_block; Status.ID:=FML_fb_timeout;
	Done					:= TRUE;
	Step					:= 30;
END_IF

// this function block is not usable with SFC-DC and MTR-DCI
IF Execute 
	AND	((FML_REF.DeviceType = SFC_DC)
	OR (FML_REF.DeviceType = MTR_DCI)) THEN
		Done				:= TRUE;
		Status.Err:=TRUE; Status.Cat:=FML_function_block; Status.ID:=FML_wrong_device;
		Step				:= 100;
END_IF

IF Param[1].PNU = 0 THEN
  FOR ixPar:=1 TO maxParamCount DO
    Param[ixPar].PNU 		:= listPNU[ixPar]; 			// fill in the PNU
    Param[ixPar].SUBINDEX 	:= 1;         				// fill in a fix subindex
	END_FOR
    // 1 =  540.1: Paramter Direktbetrieb Basisgeschwindigkeit directmode positioning
    // 2 =  541.1: Paramter Beschleunigung directmode positioning
    // 3 =  542.1: Paramter Verzögerung directmode positioning
END_IF;

(* ===== logic part ================================================= *)
IF NOT Execute AND (Step <> 0) THEN   					// aborting FB
	FML_REF.MemberID		:= 0;
	FML_REF.ReqID        	:= FML_FPC_REQ_none;
	FML_REF.PNU       		:= 0;
	FML_REF.Subindex   		:= 0;
	FML_REF.Value			:= 0;
	ActVelocity				:= 0;
	ActAcceleration			:= 0;
	ActDeceleration			:= 0;
 	Step                    := 0;
END_IF

CASE Step OF
  0:(* *)
  Done						:= FALSE;
  TimeStart					:= FALSE;
  Status.Err:=FALSE; Status.Cat:=FML_no_category; Status.ID:=FML_no_error;

	IF (FML_REF.MemberID = 0) AND Execute THEN 	
		Status.Err:=FALSE; Status.Cat:=FML_function_block; Status.ID:=FML_fb_busy;
		
		IF (FML_REF.DeviceType = CMMP_AS) 
		OR (FML_REF.DeviceType = CMMS_AS) 
		OR (FML_REF.DeviceType = CMMS_ST)
		OR (FML_REF.DeviceType = CMMD_AS) THEN					(* CMMP-AS or CMMS_AS or CMMS_ST or CMMD_AS *)	
			FML_REF.FPCC_Modus 	:= E_FML_FPC_MODUS.FML_FPC_MODUS_PNU_11BIT;
		ELSE 												(*******EMCA-EC or CMMO-ST*******)	
			FML_REF.FPCC_Modus 	:= E_FML_FPC_MODUS.FML_FPC_MODUS_PNU_16BIT;
		END_IF
    	FML_REF.MemberID		:= lMemberID;
		FML_REF.ReqID			:= FML_FPC_REQ_none;
		FML_REF.PNU				:= 0;
		FML_REF.Subindex		:= 0;
		FML_REF.Value			:= 0;
		ixPar					:= 1;  						// set to 1st array element
		(* writing *)
		IF Write THEN
			Param[1].Value		:= Velocity;
			Param[2].Value		:= Acceleration;
			Param[3].Value		:= Deceleration;
			Step				:= 10;
		(* reading *)
		ELSE
			Step				:= 20;
		END_IF
	ELSIF (FML_REF.MemberID <> lMemberId) AND Execute THEN
		Status.Err:=FALSE; Status.Cat:=FML_function_block; Status.ID:=FML_other_fb_active;
	END_IF

  10:(* writing parameter[ixPar] *)
  	TimeStart					:= TRUE;
	IF NOT FML_REF.Done THEN
		TimeStart				:= FALSE;  
		FML_REF.ReqID			:= FML_FPC_REQ_write_array_dword;
		FML_REF.PNU				:= Param[ixPar].PNU;
		FML_REF.Subindex		:= Param[ixPar].SUBINDEX;
		FML_REF.Value			:= Param[ixPar].VALUE;
		Step					:= 11;
	END_IF

  11:(* *)
  	TimeStart					:= TRUE;
	IF FML_REF.Done AND NOT FML_REF.Err THEN
		TimeStart				:= FALSE;
		FML_REF.ReqID			:= FML_FPC_REQ_none;
		ixPar					:= ixPar +1;
		Step					:= 10;
		IF ixPar > maxParamCount THEN
		  	Done					:= TRUE;
		  	ActVelocity			:= Param[1].VALUE;
			ActAcceleration		:= Param[2].VALUE;
			ActDeceleration		:= Param[3].VALUE;
		  	Status.Err:=FALSE; Status.Cat:=FML_no_category; Status.ID:=FML_no_error;
		  	Step				:= 30;
		END_IF
	ELSIF FML_REF.Done AND FML_REF.Err THEN
		TimeStart				:= FALSE; 
		Done					:= TRUE;
		Status.Err:=TRUE; Status.Cat:=FML_parameter_transfer; Status.ID:=FML_REF.ActValue;
		Step					:= 30;
	END_IF

  20: (* reading *)
  	TimeStart					:= TRUE;
	IF NOT FML_REF.Done THEN
		TimeStart				:= FALSE;
		FML_REF.ReqID			:= FML_FPC_REQ_read_array;
 		FML_REF.PNU				:= Param[ixPar].PNU;
 		FML_REF.Subindex		:= Param[ixPar].SUBINDEX;
 		Step					:= 21;
	END_IF

  21:(* set ouput variables*)
  	TimeStart					:= TRUE;
	IF FML_REF.Done AND NOT FML_REF.Err THEN
		TimeStart				:= FALSE;  
		FML_REF.ReqID			:= FML_FPC_REQ_none;
		Param[ixPar].Value		:= FML_REF.ActValue;
		ixPar					:= ixPar +1;
		Step					:= 20;
		IF ixPar > maxParamCount THEN
			ActVelocity			:= Param[1].VALUE;
			ActAcceleration		:= Param[2].VALUE;
			ActDeceleration		:= Param[3].VALUE;
			Done				:= TRUE;
			Status.Err:=FALSE; Status.Cat:=FML_no_category; Status.ID:=FML_no_error;
			Step				:= 30;
		END_IF
	ELSIF FML_REF.Done AND FML_REF.Err THEN
		TimeStart				:= FALSE;  
		Done					:= TRUE;
		Status.Err:=TRUE; Status.Cat:=FML_parameter_transfer; Status.ID:=FML_REF.ActValue;
		Step					:= 30;
	END_IF

  30: (* done - do nothing *)
	  ;
	  
END_CASE;

Status.Msg				:= GetStatusMessage(Status);
Error					:= Status.Err;

(* ===== end of function block ============================= *)

END_FUNCTION_BLOCK

// VISU/VIS_FPC_PNU
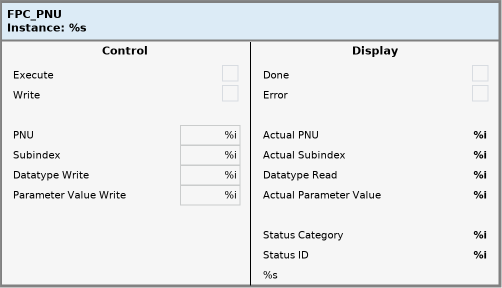
VISUALIZATION VIS_FPC_PNU  // 502x288
VAR_INPUT
	{attribute 'parameterstringof' := 'm_Input_INST'}
	m_Input_INST_Str 	: STRING;
END_VAR
VAR_IN_OUT
	m_Input_INST 		: FPC_PNU;
END_VAR
    Rectangle (0,1 500x285)
    Rectangle (0,1 500x40), "FPC_PNU Instance: %s", text variable: m_Input_INST_Str
    Rectangle (260,265 240x20), "%s", text variable: m_Input_INST.Status.Msg
    Rectangle (180,125 60x20), "%i", text variable: m_Input_INST.PNU
        OnMouseDown: write the text variable via Edit
    Rectangle (180,165 60x20), "%i", text variable: m_Input_INST.DatatypeWR
        OnMouseDown: write the text variable via Edit
    Rectangle (430,125 60x20), "%i", text variable: m_Input_INST.ActPNU
    Label (10,65 120x20), "Execute"
    Label (10,85 120x20), "Write"
    RoundedRectangle (222,65 16x16), colour toggle: m_Input_INST.Execute
        toggle m_Input_INST.Execute
    RoundedRectangle (222,85 16x16), colour toggle: m_Input_INST.Write
        toggle m_Input_INST.Write
    Label (10,125 120x20), "PNU"
    Label (10,165 120x20), "Datatype Write"
    Label (260,65 120x20), "Done"
    Label (260,85 120x20), "Error"
    RoundedRectangle (472,65 16x16), colour toggle: m_Input_INST.Done
    RoundedRectangle (472,85 16x16), colour toggle: m_Input_INST.Error
    Label (260,125 128x20), "Actual PNU"
    Label (0,41 250x20), "Control"
    Label (250,41 250x20), "Display"
    Line (250,42) (250,285)
    Rectangle (430,165 60x20), "%i", text variable: m_Input_INST.DatatypeRD
    Label (260,165 128x20), "Datatype Read"
    Rectangle (180,145 60x20), "%i", text variable: m_Input_INST.Subindex
        OnMouseDown: write the text variable via Edit
    Rectangle (430,145 60x20), "%i", text variable: m_Input_INST.ActSubindex
    Label (10,145 120x20), "Subindex"
    Label (260,145 128x20), "Actual Subindex"
    Rectangle (430,225 60x20), "%i", text variable: m_Input_INST.Status.Cat
    Label (260,225 128x20), "Status Category"
    Rectangle (430,245 60x20), "%i", text variable: m_Input_INST.Status.ID
    Label (260,245 128x20), "Status ID"
    Rectangle (180,185 60x20), "%i", text variable: m_Input_INST.Value
        OnMouseDown: write the text variable via Edit
    Label (10,185 120x20), "Parameter Value Write"
    Rectangle (430,185 60x20), "%i", text variable: m_Input_INST.ActValue
    Label (260,185 128x20), "Actual Parameter Value"
END_VISUALIZATION

// VISU/VIS_FPC_DIAG_BUFFER
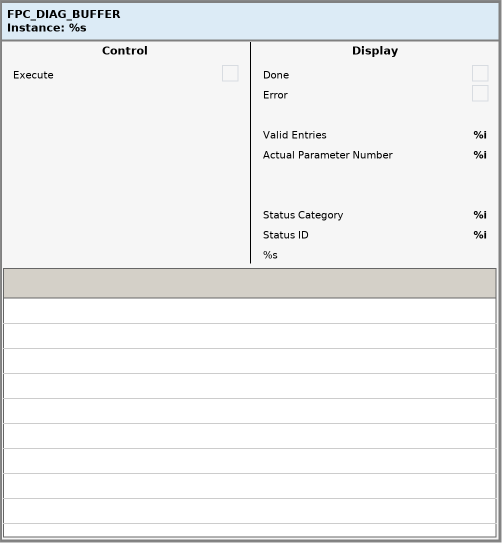
VISUALIZATION VIS_FPC_DIAG_BUFFER  // 502x543
VAR_INPUT
	{attribute 'parameterstringof' := 'm_Input_INST'}
	m_Input_INST_Str 	: STRING;
END_VAR
VAR_IN_OUT
	m_Input_INST 		: FPC_DIAG_BUFFER;
END_VAR
    Rectangle (0,1 500x540)
    Rectangle (0,1 500x40), "FPC_DIAG_BUFFER Instance: %s", text variable: m_Input_INST_Str
    Rectangle (260,245 240x20), "%s", text variable: m_Input_INST.Status.Msg
    Rectangle (430,145 60x20), "%i", text variable: m_Input_INST.ParamNo
    Label (10,65 120x20), "Execute"
    RoundedRectangle (222,65 16x16), colour toggle: m_Input_INST.Execute
        toggle m_Input_INST.Execute
    Label (260,65 120x20), "Done"
    Label (260,85 120x20), "Error"
    RoundedRectangle (472,65 16x16), colour toggle: m_Input_INST.Done
    RoundedRectangle (472,85 16x16), colour toggle: m_Input_INST.Error
    Label (260,145 140x20), "Actual Parameter Number"
    Label (0,41 250x20), "Control"
    Label (250,41 250x20), "Display"
    Line (250,42) (250,263)
    Rectangle (430,205 60x20), "%i", text variable: m_Input_INST.Status.Cat
    Label (260,205 128x20), "Status Category"
    Rectangle (430,225 60x20), "%i", text variable: m_Input_INST.Status.ID
    Label (260,225 128x20), "Status ID"
    Rectangle (430,125 60x20), "%i", text variable: m_Input_INST.ValidEntries
    Label (260,125 140x20), "Valid Entries"
    Table (3,268 493x269), data array: m_Input_INST.astVisu
        p3854506369: m_Input_INST.astVisu[INDEX].sEvent
        p1892666644: m_Input_INST.astVisu[INDEX].sStamp
        p338671338: m_Input_INST.astVisu[INDEX].sFault
        p2170511999: m_Input_INST.astVisu[INDEX].sText
        p511219082: TimeStamp
        p1755163831: Message #
        p4092479075: Message Description
END_VISUALIZATION

// VISU/VIS_FPC_DIRMP
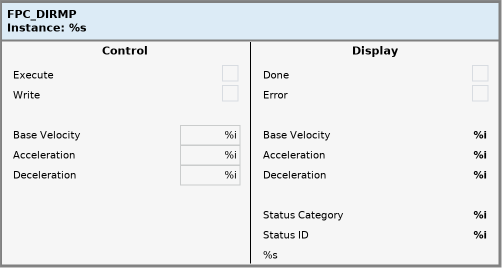
VISUALIZATION VIS_FPC_DIRMP  // 502x268
VAR_INPUT
	{attribute 'parameterstringof' := 'm_Input_INST'}
	m_Input_INST_Str 	: STRING;
END_VAR
VAR_IN_OUT
	m_Input_INST 		: FPC_DIRMP;
END_VAR
    Rectangle (0,1 500x265)
    Rectangle (0,1 500x40), "FPC_DIRMP Instance: %s", text variable: m_Input_INST_Str
    Rectangle (260,245 240x20), "%s", text variable: m_Input_INST.Status.Msg
    Rectangle (180,125 60x20), "%i", text variable: m_Input_INST.Velocity
        OnMouseDown: write the text variable via Edit
    Rectangle (180,165 60x20), "%i", text variable: m_Input_INST.Deceleration
        OnMouseDown: write the text variable via Edit
    Rectangle (430,125 60x20), "%i", text variable: m_Input_INST.ActVelocity
    Label (10,65 120x20), "Execute"
    Label (10,85 120x20), "Write"
    RoundedRectangle (222,65 16x16), colour toggle: m_Input_INST.Execute
        toggle m_Input_INST.Execute
    RoundedRectangle (222,85 16x16), colour toggle: m_Input_INST.Write
        toggle m_Input_INST.Write
    Label (10,125 120x20), "Base Velocity"
    Label (10,165 120x20), "Deceleration"
    Label (260,65 120x20), "Done"
    Label (260,85 120x20), "Error"
    RoundedRectangle (472,65 16x16), colour toggle: m_Input_INST.Done
    RoundedRectangle (472,85 16x16), colour toggle: m_Input_INST.Error
    Label (260,125 128x20), "Base Velocity"
    Label (0,41 250x20), "Control"
    Label (250,41 250x20), "Display"
    Line (250,42) (250,263)
    Rectangle (430,165 60x20), "%i", text variable: m_Input_INST.ActDeceleration
    Label (260,165 128x20), "Deceleration"
    Rectangle (180,145 60x20), "%i", text variable: m_Input_INST.Acceleration
        OnMouseDown: write the text variable via Edit
    Rectangle (430,145 60x20), "%i", text variable: m_Input_INST.ActAcceleration
    Label (10,145 120x20), "Acceleration"
    Label (260,145 128x20), "Acceleration"
    Rectangle (430,205 60x20), "%i", text variable: m_Input_INST.Status.Cat
    Label (260,205 128x20), "Status Category"
    Rectangle (430,225 60x20), "%i", text variable: m_Input_INST.Status.ID
    Label (260,225 128x20), "Status ID"
END_VISUALIZATION

// VISU/VIS_FPC_DATA_OBJECT
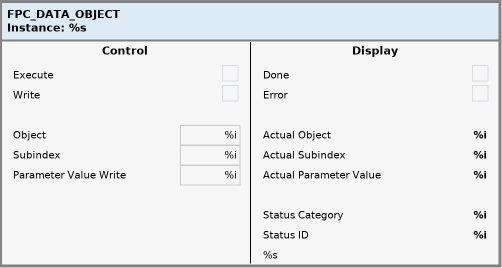
VISUALIZATION VIS_FPC_DATA_OBJECT  // 502x268
VAR_INPUT
	{attribute 'parameterstringof' := 'm_Input_INST'}
	m_Input_INST_Str	: STRING;
END_VAR
VAR_IN_OUT
	m_Input_INST 		: FPC_DATA_OBJECT;
END_VAR
    Rectangle (0,1 500x265)
    Rectangle (0,1 500x40), "FPC_DATA_OBJECT Instance: %s", text variable: m_Input_INST_Str
    Rectangle (260,245 240x20), "%s", text variable: m_Input_INST.Status.Msg
    Rectangle (180,125 60x20), "%i", text variable: m_Input_INST.Object
        OnMouseDown: write the text variable via Edit
    Rectangle (180,165 60x20), "%i", text variable: m_Input_INST.Value
        OnMouseDown: write the text variable via Edit
    Rectangle (430,125 60x20), "%i", text variable: m_Input_INST.ActObject
    Label (10,65 120x20), "Execute"
    Label (10,85 120x20), "Write"
    RoundedRectangle (222,65 16x16), colour toggle: m_Input_INST.Execute
        toggle m_Input_INST.Execute
    RoundedRectangle (222,85 16x16), colour toggle: m_Input_INST.Write
        toggle m_Input_INST.Write
    Label (10,125 120x20), "Object"
    Label (10,165 120x20), "Parameter Value Write"
    Label (260,65 120x20), "Done"
    Label (260,85 120x20), "Error"
    RoundedRectangle (472,65 16x16), colour toggle: m_Input_INST.Done
    RoundedRectangle (472,85 16x16), colour toggle: m_Input_INST.Error
    Label (260,125 128x20), "Actual Object"
    Label (0,41 250x20), "Control"
    Label (250,41 250x20), "Display"
    Line (250,42) (250,263)
    Rectangle (430,165 60x20), "%i", text variable: m_Input_INST.ActValue
    Label (260,165 128x20), "Actual Parameter Value"
    Rectangle (180,145 60x20), "%i", text variable: m_Input_INST.Subindex
        OnMouseDown: write the text variable via Edit
    Rectangle (430,145 60x20), "%i", text variable: m_Input_INST.ActSubindex
    Label (10,145 120x20), "Subindex"
    Label (260,145 128x20), "Actual Subindex"
    Rectangle (430,205 60x20), "%i", text variable: m_Input_INST.Status.Cat
    Label (260,205 128x20), "Status Category"
    Rectangle (430,225 60x20), "%i", text variable: m_Input_INST.Status.ID
    Label (260,225 128x20), "Status ID"
END_VISUALIZATION

// VISU/VIS_FHPP_CTRL
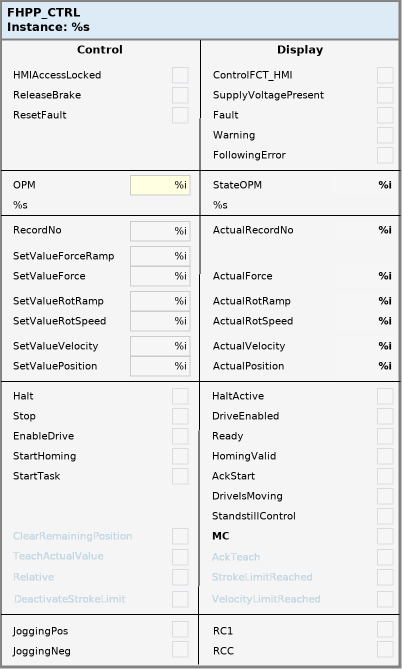
VISUALIZATION VIS_FHPP_CTRL  // 402x669
VAR_INPUT
	{attribute 'parameterstringof' := 'm_Input_INST'}
	m_Input_INST_Str 	: STRING;
END_VAR
VAR_IN_OUT
	m_Input_INST 		: FHPP_CTRL;
END_VAR
    Rectangle (0,1 400x666)
    Rectangle (0,0 400x40), "FHPP_CTRL Instance: %s", text variable: m_Input_INST_Str
    Rectangle (10,195 180x20), "%s", text variable: m_Input_INST.OPMString
    Rectangle (130,266 60x20), "%i", text variable: m_Input_INST.SetValueForce, colour toggle: (m_Input_INST.OPM) = 5
        OnMouseDown: write the text variable via Edit
    Rectangle (330,175 65x20), "%i", text variable: m_Input_INST.StateOPM
    Rectangle (130,336 60x20), "%i", tooltip "permissible range of value is 0 to 100", text variable: m_Input_INST.SetValueVelocity, colour toggle: (m_Input_INST.OPM= 1) or ((m_Input_INST.OPM =5) AND (m_Input_INST.tempVisuMode =2))
        OnMouseDown: write the text variable via Edit
    Rectangle (335,336 60x20), "%i", text variable: m_Input_INST.ActualVelocity, colour toggle: (m_Input_INST.StateOPM) = 1
    Rectangle (130,291 60x20), "%i", tooltip "permissible range of value is 0 to 100", text variable: m_Input_INST.SetValueRotRamp, colour toggle: m_Input_INST.OPM = 9
        OnMouseDown: write the text variable via Edit
    Rectangle (335,291 60x20), "%i", text variable: m_Input_INST.ActualRotRamp, colour toggle: (m_Input_INST.StateOPM) = 9
    Rectangle (130,311 60x20), "%i", text variable: m_Input_INST.SetValueRotSpeed, colour toggle: (m_Input_INST.OPM) = 9
        OnMouseDown: write the text variable via Edit
    Rectangle (335,311 60x20), "%i", text variable: m_Input_INST.ActualRotSpeed, colour toggle: (m_Input_INST.StateOPM) = 9
    Rectangle (130,356 60x20), "%i", text variable: m_Input_INST.SetValuePosition, colour toggle: (m_Input_INST.OPM) = 1
        OnMouseDown: write the text variable via Edit
    Rectangle (335,356 60x20), "%i", text variable: m_Input_INST.ActualPosition, colour toggle: (m_Input_INST.StateOPM = 1) or (m_Input_INST.StateOPM = 5) or (m_Input_INST.StateOPM = 0)
    Rectangle (210,195 180x20), "%s", text variable: m_Input_INST.StateOPMString
    Rectangle (335,266 60x20), "%i", text variable: m_Input_INST.ActualForce, colour toggle: (m_Input_INST.StateOPM) = 5
    Rectangle (335,220 60x20), "%i", text variable: m_Input_INST.ActualRecordNo, colour toggle: (m_Input_INST.StateOPM) = 0
    RoundedRectangle (377,428 16x16), colour toggle: m_Input_Inst.Ready
    RoundedRectangle (172,428 16x16), colour toggle: m_Input_Inst.EnableDrive
        toggle m_Input_Inst.EnableDrive
    RoundedRectangle (172,388 16x16), colour toggle: m_Input_Inst.Halt
        toggle m_Input_Inst.Halt
    RoundedRectangle (172,408 16x16), colour toggle: m_Input_Inst.Stop
        toggle m_Input_Inst.Stop
    RoundedRectangle (377,388 16x16), colour toggle: m_Input_Inst.HaltActive
    RoundedRectangle (377,408 16x16), colour toggle: m_Input_Inst.DriveEnabled
    RoundedRectangle (172,448 16x16), colour toggle: m_Input_Inst.StartHoming
        toggle m_Input_Inst.StartHoming
    RoundedRectangle (172,468 16x16), colour toggle: m_Input_Inst.StartTask
        toggle m_Input_Inst.StartTask
    RoundedRectangle (172,549 16x16), colour toggle: m_Input_Inst.TeachActualValue
        toggle m_Input_Inst.TeachActualValue
    RoundedRectangle (172,528 16x16), colour toggle: m_Input_Inst.ClearRemainingPosition
        toggle m_Input_Inst.ClearRemainingPosition
    RoundedRectangle (172,569 16x16), colour toggle: m_Input_Inst.Relative
        toggle m_Input_INST.Relative
    RoundedRectangle (377,448 16x16), colour toggle: m_Input_Inst.HomingValid
    RoundedRectangle (377,468 16x16), colour toggle: m_Input_Inst.AckStart
    RoundedRectangle (377,488 16x16), colour toggle: m_Input_Inst.DriveIsMoving
    RoundedRectangle (377,508 16x16), colour toggle: m_Input_Inst.StandstillControl
    RoundedRectangle (377,528 16x16), colour toggle: m_Input_Inst.MC
    RoundedRectangle (377,621 16x16), colour toggle: m_Input_Inst.RC1
    RoundedRectangle (377,641 16x16), colour toggle: m_Input_Inst.RCC
    Label (10,65 140x20), "HMIAccessLocked"
    Label (10,85 140x20), "ReleaseBrake"
    Label (10,105 140x20), "ResetFault"
    RoundedRectangle (172,621 16x16), colour toggle: m_Input_Inst.JoggingPos
        toggle m_Input_Inst.JoggingPos
    RoundedRectangle (172,641 16x16), colour toggle: m_Input_Inst.JoggingNeg
        toggle m_Input_Inst.JoggingNeg
    RoundedRectangle (172,67 16x16), colour toggle: m_Input_Inst.HMIAccessLocked
        toggle m_Input_Inst.HMIAccessLocked
    RoundedRectangle (172,87 16x16), colour toggle: m_Input_Inst.Brake
        toggle m_Input_Inst.Brake
    RoundedRectangle (172,107 16x16), colour toggle: m_Input_Inst.ResetFault
        toggle m_Input_Inst.ResetFault
    RoundedRectangle (377,67 16x16), colour toggle: m_Input_Inst.ControlFCT_HMI
    RoundedRectangle (377,87 16x16), colour toggle: m_Input_Inst.SupplyVoltagePresent
    RoundedRectangle (377,107 16x16), colour toggle: m_Input_Inst.Fault
    RoundedRectangle (377,127 16x16), colour toggle: m_Input_Inst.Warning
    RoundedRectangle (377,147 16x16), colour toggle: m_Input_Inst.FollowingError
    Label (210,65 120x20), "ControlFCT_HMI"
    Label (210,85 120x20), "SupplyVoltagePresent"
    Label (210,105 120x20), "Fault"
    Label (210,125 120x20), "Warning"
    Label (210,145 120x20), "FollowingError"
    Label (210,175 120x20), "StateOPM"
    Label (10,175 120x20), "OPM"
    Label (10,220 120x20), "RecordNo"
    Label (10,266 120x20), "SetValueForce"
    Label (10,291 120x20), "SetValueRotRamp"
    Label (10,311 120x20), "SetValueRotSpeed"
    Label (10,336 120x20), "SetValueVelocity"
    Label (10,356 120x20), "SetValuePosition"
    Label (10,386 120x20), "Halt"
    Label (10,406 120x20), "Stop"
    Label (10,426 120x20), "EnableDrive"
    Label (10,446 120x20), "StartHoming"
    Label (200,40 200x20), "Display"
    Label (0,40 200x20), "Control"
    Line (-1,614) (399,614)
    Line (200,40) (198,664)
    Line (0,381) (400,381)
    Line (0,215) (400,215)
    Line (0,170) (400,170)
    Label (210,220 120x20), "ActualRecordNo"
    Label (210,266 120x20), "ActualForce"
    Label (210,291 120x20), "ActualRotRamp"
    Label (210,311 120x20), "ActualRotSpeed"
    Label (210,336 120x20), "ActualVelocity"
    Label (210,356 120x20), "ActualPosition"
    Label (209,386 120x20), "HaltActive"
    Label (209,406 120x20), "DriveEnabled"
    Label (209,426 120x20), "Ready"
    Label (209,446 120x20), "HomingValid"
    Label (209,466 120x20), "AckStart"
    Label (209,486 120x20), "DriveIsMoving"
    Label (209,506 120x20), "StandstillControl"
    Label (209,526 120x20), "MC"
    Label (210,641 120x20), "RCC"
    Label (210,621 120x20), "RC1"
    Label (10,466 120x20), "StartTask"
    Label (10,621 130x20), "JoggingPos"
    Label (10,641 130x20), "JoggingNeg"
    Rectangle (130,221 60x20), "%i", text variable: m_Input_INST.RecordNo, colour toggle: (m_Input_INST.OPM) = 0
        OnMouseDown: write the text variable via Edit
    RoundedRectangle (172,591 16x16), colour toggle: m_Input_Inst.DeactivateStrokeLimit
        toggle m_Input_Inst.DeactivateStrokeLimit
    Rectangle (130,175 60x20), "%i", tooltip "0 = Record mode 1 = Direct position control 5 = Direct torque control 9 = Direct velocity control", text variable: m_Input_INST.OPM
        OnMouseDown: write the text variable via Edit
    Group (11,589 130x20)
        Label (0,0 130x20), "DeactivateStrokeLimit", invisible if: (m_Input_INST.OPM <> 5) and (m_Input_INST.OPM <> 9)
        Label (0,0 130x20), "DeactivateStrokeLimit", invisible if: (m_Input_INST.OPM = 5) or (m_Input_INST.OPM = 9)
    Group (10,546 120x20)
        Label (0,0 120x20), "TeachActualValue", invisible if: m_Input_INST.OPM <> 0
        Label (0,0 120x20), "TeachActualValue", invisible if: m_Input_INST.OPM = 0
    Group (10,567 120x20)
        Label (0,0 120x20), "Relative", invisible if: m_Input_INST.OPM <> 1
        Label (0,0 120x20), "Relative", invisible if: m_Input_INST.OPM = 1
    Group (10,526 130x20)
        Label (0,0 130x20), "ClearRemainingPosition", invisible if: (m_Input_INST.OPM <> 1) and (m_Input_INST.OPM <> 0)
        Label (0,0 130x20), "ClearRemainingPosition", invisible if: (m_Input_INST.OPM = 1) or (m_Input_INST.OPM = 0)
    RoundedRectangle (377,549 16x16), colour toggle: m_Input_Inst.AckTeach
    Group (209,547 120x20)
        Label (0,0 120x20), "AckTeach", invisible if: m_Input_INST.OPM <> 0
        Label (0,0 120x20), "AckTeach", invisible if: m_Input_INST.OPM = 0
    RoundedRectangle (377,591 16x16), colour toggle: m_Input_Inst.VelocityLimitReached
    Group (209,589 120x20)
        Label (0,0 120x20), "VelocityLimitReached", invisible if: (m_Input_INST.OPM <> 5) and (m_Input_INST.OPM <> 9)
        Label (0,0 120x20), "VelocityLimitReached", invisible if: (m_Input_INST.OPM = 5) or (m_Input_INST.OPM = 9)
    RoundedRectangle (377,569 16x16), colour toggle: m_Input_Inst.StrokeLimitReached
    Group (209,567 120x20)
        Label (0,0 120x20), "StrokeLimitReached", invisible if: (m_Input_INST.OPM <> 9) and (m_Input_INST.OPM <> 5)
        Label (0,0 120x20), "StrokeLimitReached", invisible if: (m_Input_INST.OPM = 5) or (m_Input_INST.OPM = 9)
    Rectangle (130,246 60x20), "%i", tooltip "permissible range of value is 0 to 100", text variable: m_Input_INST.SetValueForceRamp, colour toggle: (m_Input_INST.OPM = 5) AND (m_Input_INST.tempVisuMode =1)
        OnMouseDown: write the text variable via Edit
    Label (10,246 120x20), "SetValueForceRamp"
END_VISUALIZATION

// VISU/VIS_FPC_DIAG
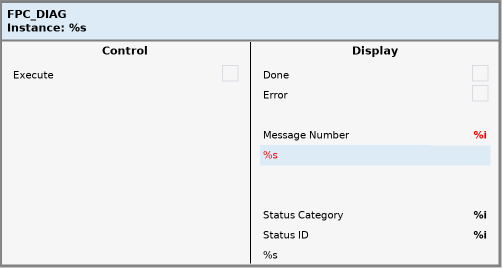
VISUALIZATION VIS_FPC_DIAG  // 502x268
VAR_INPUT
	{attribute 'parameterstringof' := 'm_Input_INST'}
	m_Input_INST_Str 	: STRING;
END_VAR
VAR_IN_OUT
	m_Input_INST 		: FPC_DIAG;
END_VAR
    Rectangle (0,1 500x265)
    Rectangle (0,1 500x40), "FPC_DIAG Instance: %s", text variable: m_Input_INST_Str
    Rectangle (260,245 240x20), "%s", text variable: m_Input_INST.Status.Msg
    Label (10,65 120x20), "Execute"
    RoundedRectangle (222,65 16x16), colour toggle: m_Input_INST.Execute
        toggle m_Input_INST.Execute
    Label (260,65 120x20), "Done"
    Label (260,85 120x20), "Error"
    RoundedRectangle (472,65 16x16), colour toggle: m_Input_INST.Done
    RoundedRectangle (472,85 16x16), colour toggle: m_Input_INST.Error
    Label (260,125 128x20), "Message Number"
    Label (0,41 250x20), "Control"
    Label (250,41 250x20), "Display"
    Line (250,42) (250,263)
    Rectangle (430,205 60x20), "%i", text variable: m_Input_INST.Status.Cat
    Label (260,205 128x20), "Status Category"
    Rectangle (430,225 60x20), "%i", text variable: m_Input_INST.Status.ID
    Label (260,225 128x20), "Status ID"
    Rectangle (260,145 230x20), "%s", text variable: m_Input_INST.MessageDescription
    Rectangle (430,125 60x20), "%i", text variable: m_Input_INST.MessageNumber
END_VISUALIZATION

// VISU/VIS_FPC_MULTI
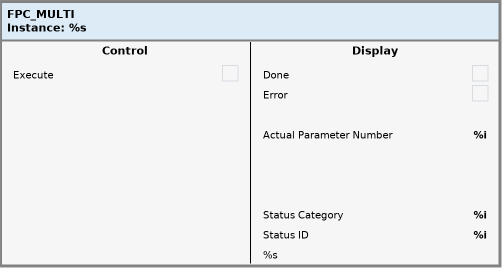
VISUALIZATION VIS_FPC_MULTI  // 502x268
VAR_INPUT
	{attribute 'parameterstringof' := 'm_Input_INST'}
	m_Input_INST_Str 	: STRING;
END_VAR
VAR_IN_OUT
	m_Input_INST 		: FPC_MULTI;
END_VAR
    Rectangle (0,1 500x265)
    Rectangle (0,1 500x40), "FPC_MULTI Instance: %s", text variable: m_Input_INST_Str
    Rectangle (260,245 240x20), "%s", text variable: m_Input_INST.Status.Msg
    Rectangle (430,125 60x20), "%i", text variable: m_Input_INST.ParamNo
    Label (10,65 120x20), "Execute"
    RoundedRectangle (222,65 16x16), colour toggle: m_Input_INST.Execute
        toggle m_Input_INST.Execute
    Label (260,65 120x20), "Done"
    Label (260,85 120x20), "Error"
    RoundedRectangle (472,65 16x16), colour toggle: m_Input_INST.Done
    RoundedRectangle (472,85 16x16), colour toggle: m_Input_INST.Error
    Label (260,125 140x20), "Actual Parameter Number"
    Label (0,41 250x20), "Control"
    Label (250,41 250x20), "Display"
    Line (250,42) (250,263)
    Rectangle (430,205 60x20), "%i", text variable: m_Input_INST.Status.Cat
    Label (260,205 128x20), "Status Category"
    Rectangle (430,225 60x20), "%i", text variable: m_Input_INST.Status.ID
    Label (260,225 128x20), "Status ID"
END_VISUALIZATION

// VISU/VIS_FPC_FILE_ARRAY
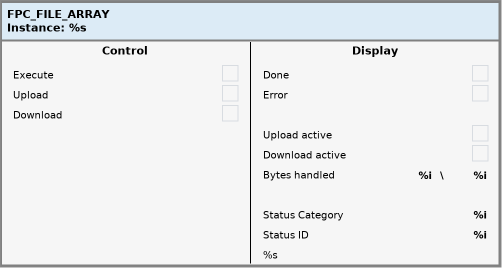
VISUALIZATION VIS_FPC_FILE_ARRAY  // 502x268
VAR_INPUT
	{attribute 'parameterstringof' := 'm_Input_INST'}
	m_Input_INST_Str 	: STRING;
END_VAR
VAR_IN_OUT
	m_Input_INST 		: FPC_FILE_ARRAY;
END_VAR
    Rectangle (0,1 500x265)
    Rectangle (0,1 500x40), "FPC_FILE_ARRAY Instance: %s", text variable: m_Input_INST_Str
    Rectangle (260,245 240x20), "%s", text variable: m_Input_INST.Status.Msg
    Label (10,65 120x20), "Execute"
    Label (10,85 120x20), "Upload"
    RoundedRectangle (222,65 16x16), colour toggle: m_Input_INST.Execute
        toggle m_Input_INST.Execute
    RoundedRectangle (222,85 16x16), colour toggle: m_Input_INST.Upload
        toggle m_Input_INST.Upload
    Label (260,65 120x20), "Done"
    Label (260,85 120x20), "Error"
    RoundedRectangle (472,65 16x16), colour toggle: m_Input_INST.Done
    RoundedRectangle (472,85 16x16), colour toggle: m_Input_INST.Error
    Label (0,41 250x20), "Control"
    Label (250,41 250x20), "Display"
    Line (250,42) (250,263)
    Rectangle (430,205 60x20), "%i", text variable: m_Input_INST.Status.Cat
    Label (260,205 128x20), "Status Category"
    Rectangle (430,225 60x20), "%i", text variable: m_Input_INST.Status.ID
    Label (260,225 128x20), "Status ID"
    Label (10,105 120x20), "Download"
    RoundedRectangle (222,105 16x16), colour toggle: m_Input_INST.Download
        toggle m_Input_INST.Download p2164770859=TRUE
    Rectangle (440,165 50x21), "%i", text variable: m_Input_INST.FileSize
    Label (260,125 120x20), "Upload active"
    Label (260,165 120x20), "Bytes handled"
    Label (260,145 120x20), "Download active"
    Rectangle (385,165 50x21), "%i", text variable: m_Input_INST.CountByte
    Label (437,165 13x21), "\"
    RoundedRectangle (472,125 16x16), colour toggle: m_Input_INST.vis_upload
    RoundedRectangle (472,145 16x16), colour toggle: m_Input_INST.vis_download
END_VISUALIZATION

// VISU/VIS_FHPP_CTRL_CMXH
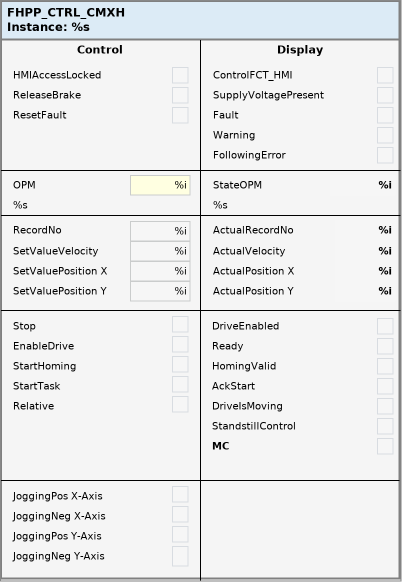
VISUALIZATION VIS_FHPP_CTRL_CMXH  // 402x582
VAR_INPUT
	{attribute 'parameterstringof' := 'm_Input_INST'}
	m_Input_INST_Str 	: STRING;
END_VAR
VAR_IN_OUT
	m_Input_INST 		: FHPP_CTRL_CMXH;
END_VAR
    Rectangle (0,0 400x579)
    Rectangle (0,0 400x40), "FHPP_CTRL_CMXH Instance: %s", text variable: m_Input_INST_Str
    Rectangle (10,195 180x20), "%s", text variable: m_Input_INST.OPMString
    Rectangle (330,175 65x20), "%i", text variable: m_Input_INST.StateOPM
    Rectangle (130,241 60x20), "%i", tooltip "permissible range of value is 0 to 100", text variable: m_Input_INST.SetValueVelocity, colour toggle: (m_Input_INST.OPM= 1) or ((m_Input_INST.OPM =5) AND (m_Input_INST.tempVisuMode =2))
        OnMouseDown: write the text variable via Edit
    Rectangle (335,241 60x20), "%i", text variable: m_Input_INST.ActualVelocity, colour toggle: (m_Input_INST.StateOPM) = 1
    Rectangle (130,261 60x20), "%i", text variable: m_Input_INST.SetValuePositionX, colour toggle: (m_Input_INST.OPM) = 1
        OnMouseDown: write the text variable via Edit
    Rectangle (335,261 60x20), "%i", text variable: m_Input_INST.ActualPositionX, colour toggle: (m_Input_INST.StateOPM = 1) or (m_Input_INST.StateOPM = 5) or (m_Input_INST.StateOPM = 0)
    Rectangle (210,195 180x20), "%s", text variable: m_Input_INST.StateOPMString
    Rectangle (335,220 60x20), "%i", text variable: m_Input_INST.ActualRecordNo, colour toggle: (m_Input_INST.StateOPM) = 0
    RoundedRectangle (377,338 16x16), colour toggle: m_Input_Inst.Ready
    RoundedRectangle (172,336 16x16), colour toggle: m_Input_Inst.EnableDrive
        toggle m_Input_Inst.EnableDrive
    RoundedRectangle (172,316 16x16), colour toggle: m_Input_Inst.Stop
        toggle m_Input_Inst.Stop
    RoundedRectangle (377,318 16x16), colour toggle: m_Input_Inst.DriveEnabled
    RoundedRectangle (172,356 16x16), colour toggle: m_Input_Inst.StartHoming
        toggle m_Input_Inst.StartHoming
    RoundedRectangle (172,376 16x16), colour toggle: m_Input_Inst.StartTask
        toggle m_Input_Inst.StartTask
    RoundedRectangle (172,396 16x16), colour toggle: m_Input_Inst.Relative
        toggle m_Input_INST.Relative
    RoundedRectangle (377,358 16x16), colour toggle: m_Input_Inst.HomingValid
    RoundedRectangle (377,378 16x16), colour toggle: m_Input_Inst.AckStart
    RoundedRectangle (377,398 16x16), colour toggle: m_Input_Inst.DriveIsMoving
    RoundedRectangle (377,418 16x16), colour toggle: m_Input_Inst.StandstillControl
    RoundedRectangle (377,438 16x16), colour toggle: m_Input_Inst.MC
    Label (10,65 140x20), "HMIAccessLocked"
    Label (10,85 140x20), "ReleaseBrake"
    Label (10,105 140x20), "ResetFault"
    RoundedRectangle (172,486 16x16), colour toggle: m_Input_INST.JogPosX
        toggle m_Input_INST.JogPosX
    RoundedRectangle (172,506 16x16), colour toggle: m_Input_Inst.JogNegX
        toggle m_Input_INST.JogNegX
    RoundedRectangle (172,67 16x16), colour toggle: m_Input_Inst.HMIAccessLocked
        toggle m_Input_Inst.HMIAccessLocked
    RoundedRectangle (172,87 16x16), colour toggle: m_Input_Inst.Brake
        toggle m_Input_Inst.Brake
    RoundedRectangle (172,107 16x16), colour toggle: m_Input_Inst.ResetFault
        toggle m_Input_Inst.ResetFault
    RoundedRectangle (377,67 16x16), colour toggle: m_Input_Inst.ControlFCT_HMI
    RoundedRectangle (377,87 16x16), colour toggle: m_Input_Inst.SupplyVoltagePresent
    RoundedRectangle (377,107 16x16), colour toggle: m_Input_Inst.Fault
    RoundedRectangle (377,127 16x16), colour toggle: m_Input_Inst.Warning
    RoundedRectangle (377,147 16x16), colour toggle: m_Input_Inst.FollowingError
    Label (210,65 120x20), "ControlFCT_HMI"
    Label (210,85 120x20), "SupplyVoltagePresent"
    Label (210,105 120x20), "Fault"
    Label (210,125 120x20), "Warning"
    Label (210,145 120x20), "FollowingError"
    Label (210,175 120x20), "StateOPM"
    Label (10,175 120x20), "OPM"
    Label (10,220 120x20), "RecordNo"
    Label (10,241 120x20), "SetValueVelocity"
    Label (10,261 120x20), "SetValuePosition X"
    Label (10,316 120x20), "Stop"
    Label (10,336 120x20), "EnableDrive"
    Label (10,356 120x20), "StartHoming"
    Label (200,40 200x20), "Display"
    Label (0,40 200x20), "Control"
    Line (-1,480) (399,480)
    Line (200,40) (200,580)
    Line (0,310) (400,310)
    Line (0,215) (400,215)
    Line (0,170) (400,170)
    Label (210,220 120x20), "ActualRecordNo"
    Label (210,241 120x20), "ActualVelocity"
    Label (210,261 120x20), "ActualPosition X"
    Label (209,316 120x20), "DriveEnabled"
    Label (209,336 120x20), "Ready"
    Label (209,356 120x20), "HomingValid"
    Label (209,376 120x20), "AckStart"
    Label (209,396 120x20), "DriveIsMoving"
    Label (209,416 120x20), "StandstillControl"
    Label (209,436 120x20), "MC"
    Label (10,376 120x20), "StartTask"
    Label (10,486 130x20), "JoggingPos X-Axis"
    Label (10,506 130x20), "JoggingNeg X-Axis"
    Rectangle (130,221 60x20), "%i", text variable: m_Input_INST.RecordNo, colour toggle: (m_Input_INST.OPM) = 0
        OnMouseDown: write the text variable via Edit
    Rectangle (130,175 60x20), "%i", tooltip "0 = Record mode 1 = Direct position control", text variable: m_Input_INST.OPM
        OnMouseDown: write the text variable via Edit
    Label (10,526 130x20), "JoggingPos Y-Axis"
    Label (10,546 130x20), "JoggingNeg Y-Axis"
    RoundedRectangle (172,526 16x16), colour toggle: m_Input_INST.JogPosY
        toggle m_Input_INST.JogPosY
    RoundedRectangle (172,546 16x20), colour toggle: m_Input_INST.JogNegY
        toggle m_Input_INST.JogNegY
    Label (10,396 120x20), "Relative"
    Label (10,281 120x20), "SetValuePosition Y"
    Rectangle (130,281 60x20), "%i", text variable: m_Input_INST.SetValuePositionY, colour toggle: (m_Input_INST.OPM) = 1
        OnMouseDown: write the text variable via Edit
    Rectangle (335,281 60x20), "%i", text variable: m_Input_INST.ActualPositionY, colour toggle: (m_Input_INST.StateOPM = 1) or (m_Input_INST.StateOPM = 5) or (m_Input_INST.StateOPM = 0)
    Label (210,281 120x20), "ActualPosition Y"
END_VISUALIZATION
